(* Local variables generated by Rascal *)
END_VAR
(* ++Tomato++CodeBlock: 06094-06096 is LogicCondition 00511.1 AND 00037.2 AND NOT 00030.0  *)
IF S_1SEC AND FASE_7 AND NOT TIMER_41 THEN (* !triggerpuls 1,0 sec. AND !fase 7 AND NOT  *)
  (* ++Lime++CodeBlock: 06097-06101 is DecrementCounter 01264,01265,01266,01267 => 00030.0  *)
  IF DSP41_0 > 0 THEN (* !display 41 eenheden *)
    DSP41_0 := DSP41_0 - 1 ;
  ELSIF DSP41_1 > 0 THEN (* !display 41 tientallen *)
    DSP41_0 := 9;
    DSP41_1 := DSP41_1 - 1 ;
  ELSIF DSP41_2 > 0 THEN (* !display 41 honderdtallen *)
    DSP41_0 := 9;
    DSP41_1 := 9;
    DSP41_2 := DSP41_2 - 1 ;
  ELSIF DSP41_3 > 0 THEN (* !display 41 duizendtallen *)
    DSP41_0 := 9;
    DSP41_1 := 9;
    DSP41_2 := 9;
    DSP41_3 := DSP41_3 - 1 ;
  ELSE (* Timer underflow, rolling over to maximum value *)
    DSP41_0 := 9;
    DSP41_1 := 9;
    DSP41_2 := 9;
    DSP41_3 := 9;
  END_IF;
  TIMER_41 := (0 = DSP41_0) AND (0 = DSP41_1) AND (0 = DSP41_2) AND (0 = DSP41_3) ; (*  *)
END_IF;
  
(* ++Tomato++CodeBlock: 06102-06102 is LogicCondition NOT 00037.2  *)
IF  NOT FASE_7 THEN (*  NOT !fase 7 *)
  (* ++Lime++CodeBlock: 06103-06110 is AssignValue 02164,02165,02166,02167 to 01264,01265,01266,01267 *)
  DSP41_0 := STP41_0 ; (* !setpoint 41 eenheden ==>> !display 41 eenheden *)
  DSP41_1 := STP41_1 ; (* !setpoint 41 tientallen ==>> !display 41 tientallen *)
  DSP41_2 := STP41_2 ; (* !setpoint 41 honderdtallen ==>> !display 41 honderdtallen *)
  DSP41_3 := STP41_3 ; (* !setpoint 41 duizendtallen ==>> !display 41 duizendtallen *)
    
  (* ++Brown++CodeBlock: 06111-06111 is ResetBit 00030.0  *)
  TIMER_41 := FALSE ; (*  *)
END_IF;
  
END_PROGRAM

(* POU IO_Mapping, ST *)
PROGRAM IO_Mapping
VAR
	bSecondPulse AT %QX256.0 : BOOL ; (**< 50% Duty cycle second pulse *)
	TriggerState AT %QX256.1 : BOOL ; (**< Trigger Condition *)
	TimerResult AT %QX256.2 : BOOL ; (**< Timer Expiration *)
	ActualCount AT %QW257 : INT ; (**< Actual count sent by modbus TCP *)
	Cycles AT %QW258  : WORD ; (**< CycleCount *)
	bEnableCount AT %IX256.0 : BOOL ; (**< Enable input received by the modbus TCP *)
	bMinutePulse AT %QX256.3 : BOOL ; (**< 50% Duty cycle minute pulse *)
	Trigger : R_TRIG ;
END_VAR
WriteBit(ADR(PC20_CYCLE.FASE_7), bEnableCount );

bSecondPulse := _CLOCK_1S ;
bMinutePulse := _CLOCK_60S ;
TriggerState := _CLOCK_1S AND PC20_CYCLE.FASE_7 AND NOT PC20_CYCLE.TIMER_41;
TimerResult := PC20_CYCLE.TIMER_41;

ActualCount := ComposeInt(PC20_CYCLE.DSP41_0, PC20_CYCLE.DSP41_1, PC20_CYCLE.DSP41_2, PC20_CYCLE.DSP41_3);

WriteValue(ADR(PC20_CYCLE.STP41_1), 1);
Trigger(CLK:= TriggerState, Q=> );
WriteBit(ADR(PC20_CYCLE.S_1SEC), Trigger.Q);

Cycles := Cycles + 1 ;
END_PROGRAM

(* POU Functions/WriteBit, ST *)
FUNCTION WriteBit : BOOL
VAR_INPUT
	pBit : POINTER TO BOOL ; (**< AddressValue of the target *)
	bValue : BOOL ; (**< Value to equalize bit to *)
END_VAR
VAR
END_VAR
pBit^ := bValue;
END_FUNCTION

(* POU Functions/ComposeInt, ST *)
FUNCTION ComposeInt : INT
VAR_INPUT
	Ones : INT ;
	Tens : INT ;
	Hundreds : INT ;
	Thousands : INT ;
END_VAR
VAR
END_VAR
ComposeInt := (Thousands * 1000) + (Hundreds * 100) + (Tens * 10) + Ones;
END_FUNCTION

(* POU Functions/WriteValue, ST *)
FUNCTION WriteValue : BOOL
VAR_INPUT
	pValue : POINTER TO INT ; (**< Pointer to value to write *)
	Value : INT ; (**< Value to store into the variable *)
END_VAR
VAR
END_VAR
pValue ^ := Value;
END_FUNCTION

(* POU Library/TTimer, ST *)
FUNCTION_BLOCK TTimer
VAR_INPUT
	Condition : BOOL ; (**< Starts the timer *)
	Setpoint : INT ; (**< Count to start *)
END_VAR

VAR_OUTPUT
	RemainingCount : INT ;
END_VAR
IF _CLOCK_1S AND Condition THEN
	RemainingCount := RemainingCount -1 ;
	IF(0 > RemainingCount) THEN
		RemainingCount := 9999;
	END_IF;
END_IF;

IF NOT Condition THEN
	RemainingCount := Setpoint;
END_IF;
END_FUNCTION_BLOCK

(* Visualisation Sample
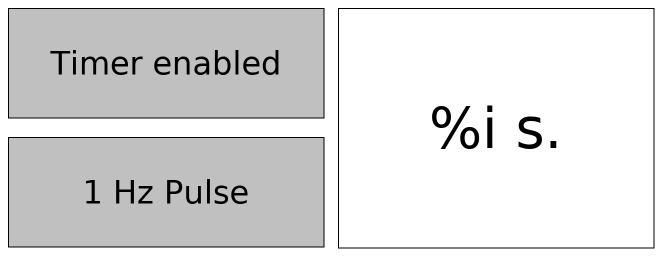
rectangle at (49,41)-(365,151): text "Timer enabled"; alarm colour if PC20_CYCLE.FASE_7
rectangle at (49,170)-(365,280): text "1 Hz Pulse"; alarm colour if ._CLOCK_1S
rectangle at (379,41)-(695,281): text "%i s."; shows IO_Mapping.ActualCount
*)
